# EPICS substitutions: llrfHlsAsynApp/Db/cableCal.substitutions
file cableCal_config.db
{
    pattern  {   DEVICE    }
             {  "$(DEV)"   }
}

file cableCal_config_raw.db
{
    pattern  {   DEVICE    }
             {  "$(DEV)"   }
}

file cableCal_mon.db
{
#                            pulse    channel
    pattern  {    DEVICE,       P,       C  }
# channel 0
             {  "$(DEV)",      "0",     "0" }
             {  "$(DEV)",      "1",     "0" }
             {  "$(DEV)",      "2",     "0" }
             {  "$(DEV)",      "3",     "0" }
# channel 1
             {  "$(DEV)",      "0",     "1" }
             {  "$(DEV)",      "1",     "1" }
             {  "$(DEV)",      "2",     "1" }
             {  "$(DEV)",      "3",     "1" }
# channel 2
             {  "$(DEV)",      "0",     "2" }
             {  "$(DEV)",      "1",     "2" }
             {  "$(DEV)",      "2",     "2" }
             {  "$(DEV)",      "3",     "2" }
# channel 3
             {  "$(DEV)",      "0",     "3" }
             {  "$(DEV)",      "1",     "3" }
             {  "$(DEV)",      "2",     "3" }
             {  "$(DEV)",      "3",     "3" }
}
